FUNCTION_BLOCK AX_MUX_3 (* AX multiplexor *)
  (* Standard: 61499-2; Description: Copyright (c) 2024 HR Agrartechnik GmbH This program and the accompanying materials are made available under the terms of the Eclipse Public License 2.0 which is available at https://www.eclipse.org/legal/epl-2.0/ SPDX-License-Identifier: EPL-2.0 *)
  (* Version 1.0, 2024-10-23, Franz Höpfinger, HR Agrartechnik GmbH *)
  PACKAGE adapter::selection::unidirectional;
  IMPORT eclipse4diac::core::TypeHash;
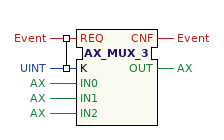
  EVENT_INPUT
    REQ WITH K; (* Set Index K *)
  END_EVENT
  EVENT_OUTPUT
    CNF; (* Confirmation of Set Index K *)
  END_EVENT
  VAR_INPUT
    K : UINT; (* index *)
  END_VAR
  SOCKETS
    IN0 : adapter::types::unidirectional::AX; (* Input value 0 *)
    IN1 : adapter::types::unidirectional::AX; (* Input value 1 *)
    IN2 : adapter::types::unidirectional::AX; (* Input value 2 *)
  END_SOCKETS
  PLUGS
    OUT : adapter::types::unidirectional::AX; (* IN0 for K = 0, IN1 for K = 1, IN2 for K = 2 *)
  END_PLUGS
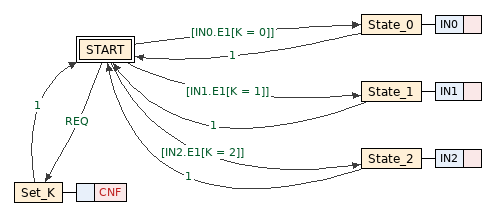
  EC_STATES
    START; (* Initial State *)
    State_0 : IN0;
    State_1 : IN1;
    Set_K : -> CNF;
    State_2 : IN2;
  END_STATES
  EC_TRANSITIONS
    START TO State_0 := [IN0.E1[K = 0]];
    START TO State_1 := [IN1.E1[K = 1]];
    State_0 TO START := 1;
    State_1 TO START := 1;
    START TO Set_K := REQ;
    Set_K TO START := 1;
    START TO State_2 := [IN2.E1[K = 2]];
    State_2 TO START := 1;
  END_TRANSITIONS
  ALGORITHM IN0 IN ST:
OUT.D1 := IN0.D1;
  END_ALGORITHM
  ALGORITHM IN1 IN ST:
OUT.D1 := IN1.D1;
  END_ALGORITHM
  ALGORITHM IN2 IN ST:
OUT.D1 := IN2.D1;
  END_ALGORITHM
END_FUNCTION_BLOCK
